FUNCTION Get_Valid_Indexs : ARRAY [1..GV_HMI.iMaxTargets] OF INT
VAR_INPUT
END_VAR
VAR
	indexes: ARRAY [1..GV_HMI.iMaxTargets] OF INT;
	i: INT;
	j: INT;
END_VAR

j := 1;
FOR i:=1 TO GV_HMI.iMaxTargets BY 1 DO 
   IF XML.savedvalues.savedpos[i].targetclear THEN
	   indexes[j] := i;
	   j := j + 1;
   END_IF
END_FOR;

Get_Valid_Indexs := indexes;

END_FUNCTION

(* stored: Version 1.1.0.1, ProductVersion 3.1.4022.12
   POU Get_Valid_Indexs: Id {a84b37d0-7817-4376-9d51-ea3cb97f205d}, SpecialFunc None *)
